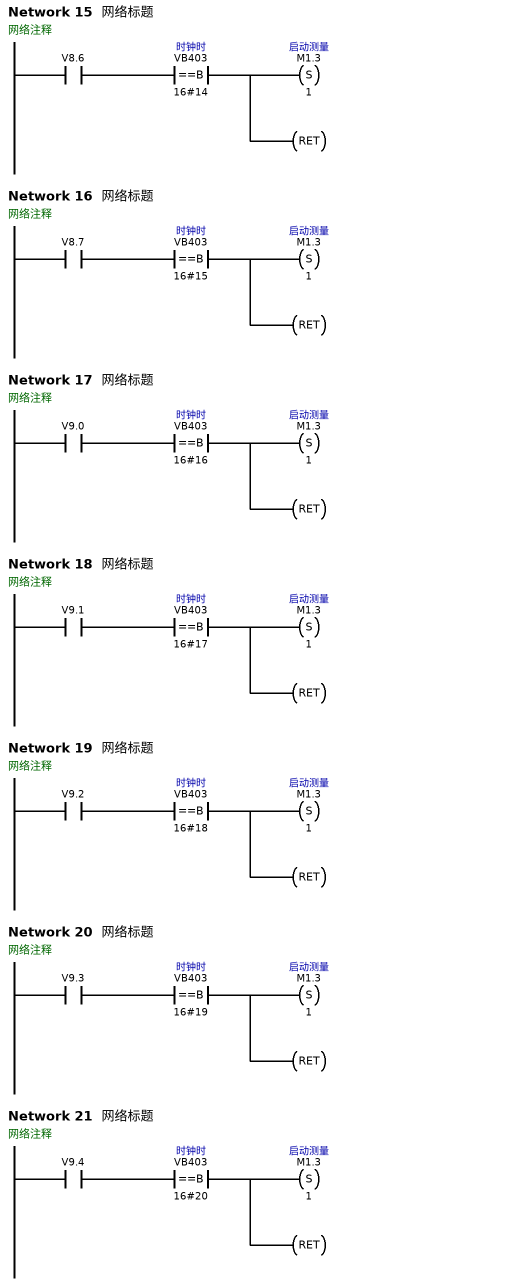
[picture p72: SBR13 networks 15-21]
Network 15 // 网络标题
// 网络注释
LD     V8.6
AB=    时钟时:VB403, 16#14
S      启动测量:M1.3, 1
CRET
Network 16 // 网络标题
// 网络注释
LD     V8.7
AB=    时钟时:VB403, 16#15
S      启动测量:M1.3, 1
CRET
Network 17 // 网络标题
// 网络注释
LD     V9.0
AB=    时钟时:VB403, 16#16
S      启动测量:M1.3, 1
CRET
Network 18 // 网络标题
// 网络注释
LD     V9.1
AB=    时钟时:VB403, 16#17
S      启动测量:M1.3, 1
CRET
Network 19 // 网络标题
// 网络注释
LD     V9.2
AB=    时钟时:VB403, 16#18
S      启动测量:M1.3, 1
CRET
Network 20 // 网络标题
// 网络注释
LD     V9.3
AB=    时钟时:VB403, 16#19
S      启动测量:M1.3, 1
CRET
Network 21 // 网络标题
// 网络注释
LD     V9.4
AB=    时钟时:VB403, 16#20
S      启动测量:M1.3, 1
CRET
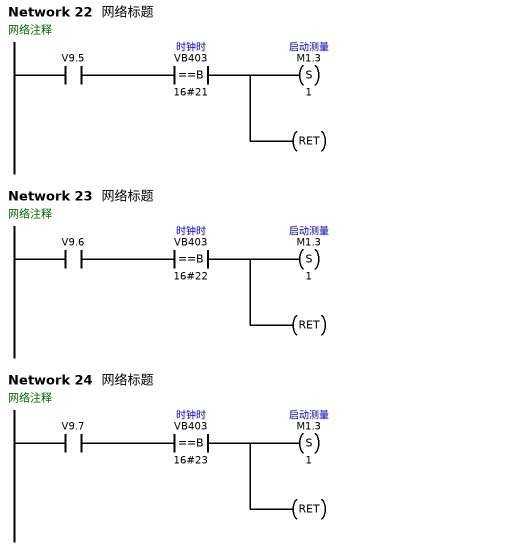
Network 22 // 网络标题
// 网络注释
LD     V9.5
AB=    时钟时:VB403, 16#21
S      启动测量:M1.3, 1
CRET
Network 23 // 网络标题
// 网络注释
LD     V9.6
AB=    时钟时:VB403, 16#22
S      启动测量:M1.3, 1
CRET
Network 24 // 网络标题
// 网络注释
LD     V9.7
AB=    时钟时:VB403, 16#23
S      启动测量:M1.3, 1
CRET
END_SUBROUTINE_BLOCK

SUBROUTINE_BLOCK Cal:SBR14
TITLE=子程序注释
VAR_INPUT
V:REAL;	// LD0 
Vo:REAL;	// LD4 
K:REAL;	// LD8 
b:REAL;	// LD12 
END_VAR
VAR_OUTPUT
吸光度:REAL;	// LD16 
值:REAL;	// LD20 
END_VAR
BEGIN
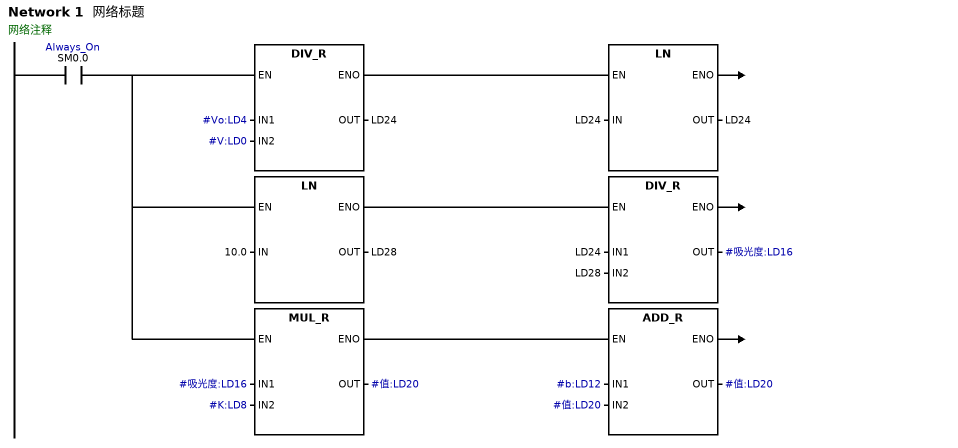
Network 1 // 网络标题
// 网络注释
LD     Always_On:SM0.0
LPS
MOVR   #Vo:LD4, LD24
AENO
/R     #V:LD0, LD24
AENO
LN     LD24, LD24
LRD
LN     10.0, LD28
AENO
MOVR   LD24, #吸光度:LD16
/R     LD28, #吸光度:LD16
LPP
MOVR   #吸光度:LD16, #值:LD20
AENO
*R     #K:LD8, #值:LD20
AENO
+R     #b:LD12, #值:LD20
END_SUBROUTINE_BLOCK

SUBROUTINE_BLOCK 偏离规则:SBR16
TITLE=子程序注释
VAR_INPUT
测量值:REAL;	// LD0 
标准值:REAL;	// LD4 
偏离比:REAL;	// LD8 0-100(10表示偏离百分之十以内视为通过)
END_VAR
VAR_OUTPUT
通过:BOOL;	// L12.0 
END_VAR
VAR
mid1:REAL;	// LD13 
mid2:REAL;	// LD17 
mid3:REAL;	// LD21 
上:REAL;	// LD25 
下:REAL;	// LD29 
END_VAR
BEGIN
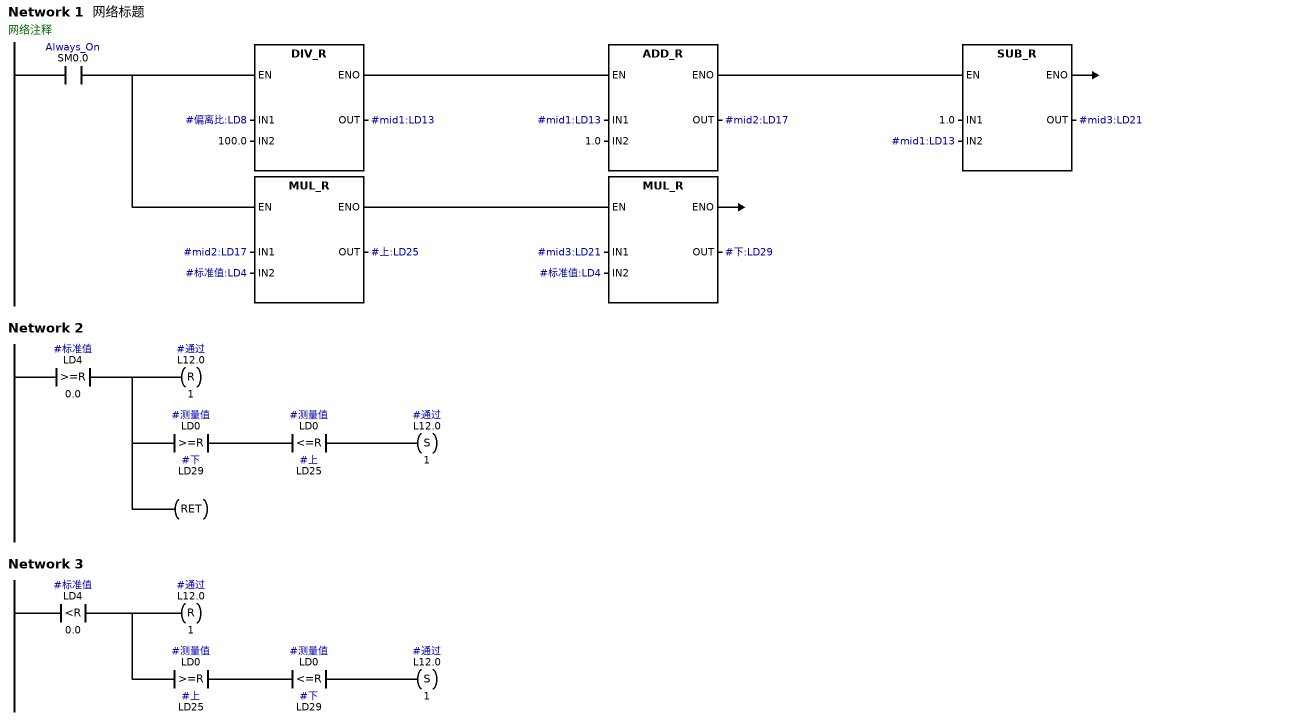
Network 1 // 网络标题
// 网络注释
LD     Always_On:SM0.0
LPS
MOVR   #偏离比:LD8, #mid1:LD13
AENO
/R     100.0, #mid1:LD13
AENO
MOVR   #mid1:LD13, #mid2:LD17
AENO
+R     1.0, #mid2:LD17
AENO
MOVR   1.0, #mid3:LD21
-R     #mid1:LD13, #mid3:LD21
LPP
MOVR   #mid2:LD17, #上:LD25
AENO
*R     #标准值:LD4, #上:LD25
AENO
MOVR   #mid3:LD21, #下:LD29
*R     #标准值:LD4, #下:LD29
Network 2
LDR>=  #标准值:LD4, 0.0
LPS
R      #通过:L12.0, 1
AR>=   #测量值:LD0, #下:LD29
AR<=   #测量值:LD0, #上:LD25
S      #通过:L12.0, 1
LPP
CRET
Network 3
LDR<   #标准值:LD4, 0.0
R      #通过:L12.0, 1
AR>=   #测量值:LD0, #上:LD25
AR<=   #测量值:LD0, #下:LD29
S      #通过:L12.0, 1
END_SUBROUTINE_BLOCK

SUBROUTINE_BLOCK 数据库:SBR17
TITLE=子程序注释
BEGIN
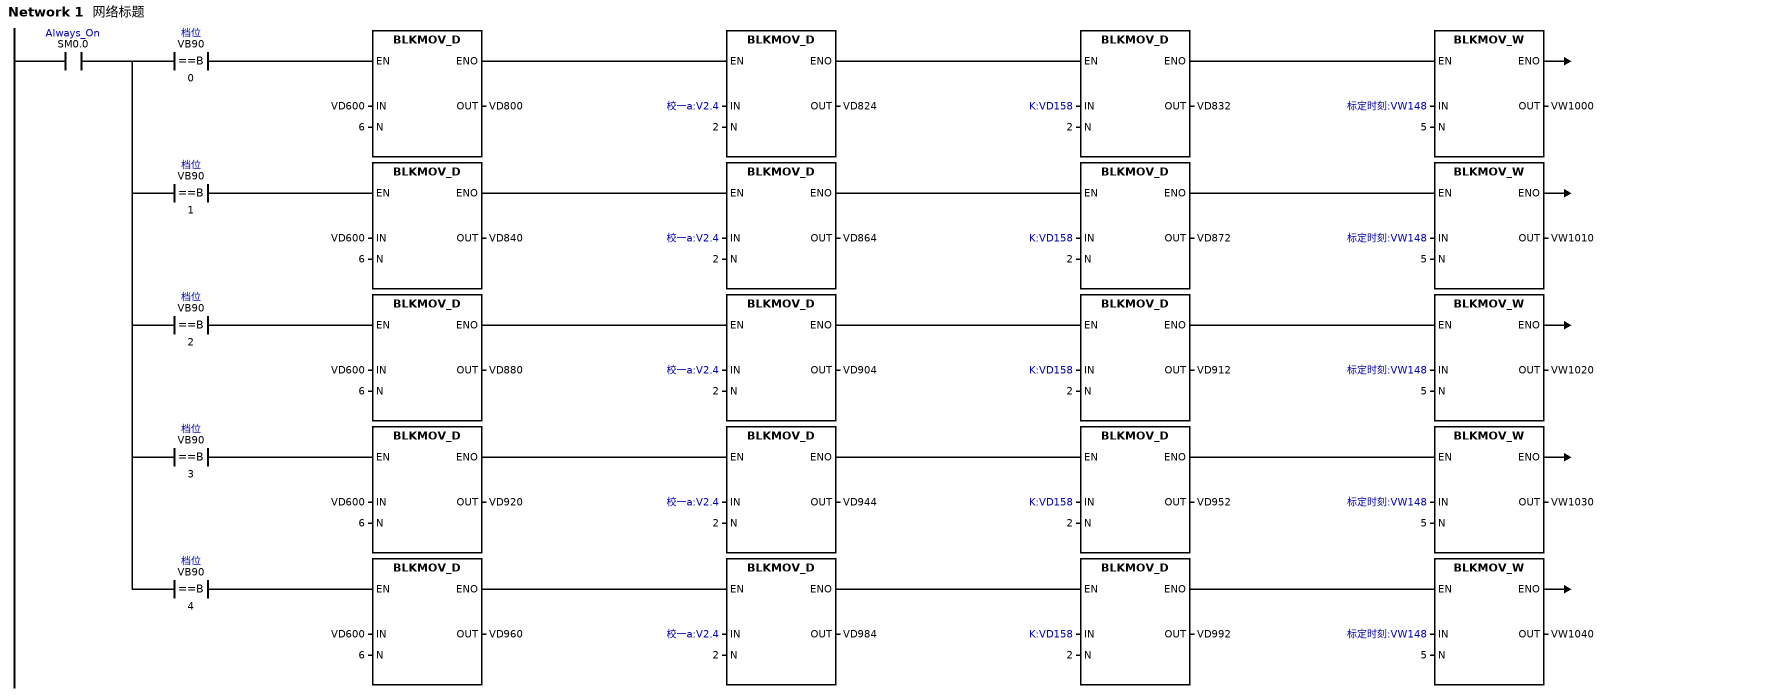
Network 1 // 网络标题
// (network saved uncompiled; LAD cells follow)
// row 0: c0 -| |- Always_On:SM0.0 v  c1 -|==B|- 档位:VB90, 0  c2 --  c3 [BLKMOV_D EN:=power@row0, IN:=VD600, N:=6, ENO=>power, OUT=>VD800]  c4 --  c5 --  c6 [BLKMOV_D EN:=power@row0, IN:=校一a:V2.4, N:=2, ENO=>power, OUT=>VD824]  c7 --  c8 --  c9 [BLKMOV_D EN:=power@row0, IN:=K:VD158, N:=2, ENO=>power, OUT=>VD832]  c10 --  c11 --  c12 [BLKMOV_W EN:=power@row0, IN:=标定时刻:VW148, N:=5, ENO=>power, OUT=>VW1000]  c13 ->
// row 1: c0 ^v  c3 [box]  c6 [box]  c9 [box]  c12 [box]
// row 2: c0 ^v  c1 -|==B|- 档位:VB90, 1  c2 --  c3 [BLKMOV_D EN:=power@row2, IN:=VD600, N:=6, ENO=>power, OUT=>VD840]  c4 --  c5 --  c6 [BLKMOV_D EN:=power@row2, IN:=校一a:V2.4, N:=2, ENO=>power, OUT=>VD864]  c7 --  c8 --  c9 [BLKMOV_D EN:=power@row2, IN:=K:VD158, N:=2, ENO=>power, OUT=>VD872]  c10 --  c11 --  c12 [BLKMOV_W EN:=power@row2, IN:=标定时刻:VW148, N:=5, ENO=>power, OUT=>VW1010]  c13 ->
// row 3: c0 ^v  c3 [box]  c6 [box]  c9 [box]  c12 [box]
// row 4: c0 ^v  c1 -|==B|- 档位:VB90, 2  c2 --  c3 [BLKMOV_D EN:=power@row4, IN:=VD600, N:=6, ENO=>power, OUT=>VD880]  c4 --  c5 --  c6 [BLKMOV_D EN:=power@row4, IN:=校一a:V2.4, N:=2, ENO=>power, OUT=>VD904]  c7 --  c8 --  c9 [BLKMOV_D EN:=power@row4, IN:=K:VD158, N:=2, ENO=>power, OUT=>VD912]  c10 --  c11 --  c12 [BLKMOV_W EN:=power@row4, IN:=标定时刻:VW148, N:=5, ENO=>power, OUT=>VW1020]  c13 ->
// row 5: c0 ^v  c3 [box]  c6 [box]  c9 [box]  c12 [box]
// row 6: c0 ^v  c1 -|==B|- 档位:VB90, 3  c2 --  c3 [BLKMOV_D EN:=power@row6, IN:=VD600, N:=6, ENO=>power, OUT=>VD920]  c4 --  c5 --  c6 [BLKMOV_D EN:=power@row6, IN:=校一a:V2.4, N:=2, ENO=>power, OUT=>VD944]  c7 --  c8 --  c9 [BLKMOV_D EN:=power@row6, IN:=K:VD158, N:=2, ENO=>power, OUT=>VD952]  c10 --  c11 --  c12 [BLKMOV_W EN:=power@row6, IN:=标定时刻:VW148, N:=5, ENO=>power, OUT=>VW1030]  c13 ->
// row 7: c0 ^v  c3 [box]  c6 [box]  c9 [box]  c12 [box]
// row 8: c0 ^  c1 -|==B|- 档位:VB90, 4  c2 --  c3 [BLKMOV_D EN:=power@row8, IN:=VD600, N:=6, ENO=>power, OUT=>VD960]  c4 --  c5 --  c6 [BLKMOV_D EN:=power@row8, IN:=校一a:V2.4, N:=2, ENO=>power, OUT=>VD984]  c7 --  c8 --  c9 [BLKMOV_D EN:=power@row8, IN:=K:VD158, N:=2, ENO=>power, OUT=>VD992]  c10 --  c11 --  c12 [BLKMOV_W EN:=power@row8, IN:=标定时刻:VW148, N:=5, ENO=>power, OUT=>VW1040]  c13 ->
// row 9: c3 [box]  c6 [box]  c9 [box]  c12 [box]
END_SUBROUTINE_BLOCK

SUBROUTINE_BLOCK 换挡:SBR19
TITLE=每个切换范围包含高低两个档位，当前处于低档则切换到高档，反之亦然
BEGIN
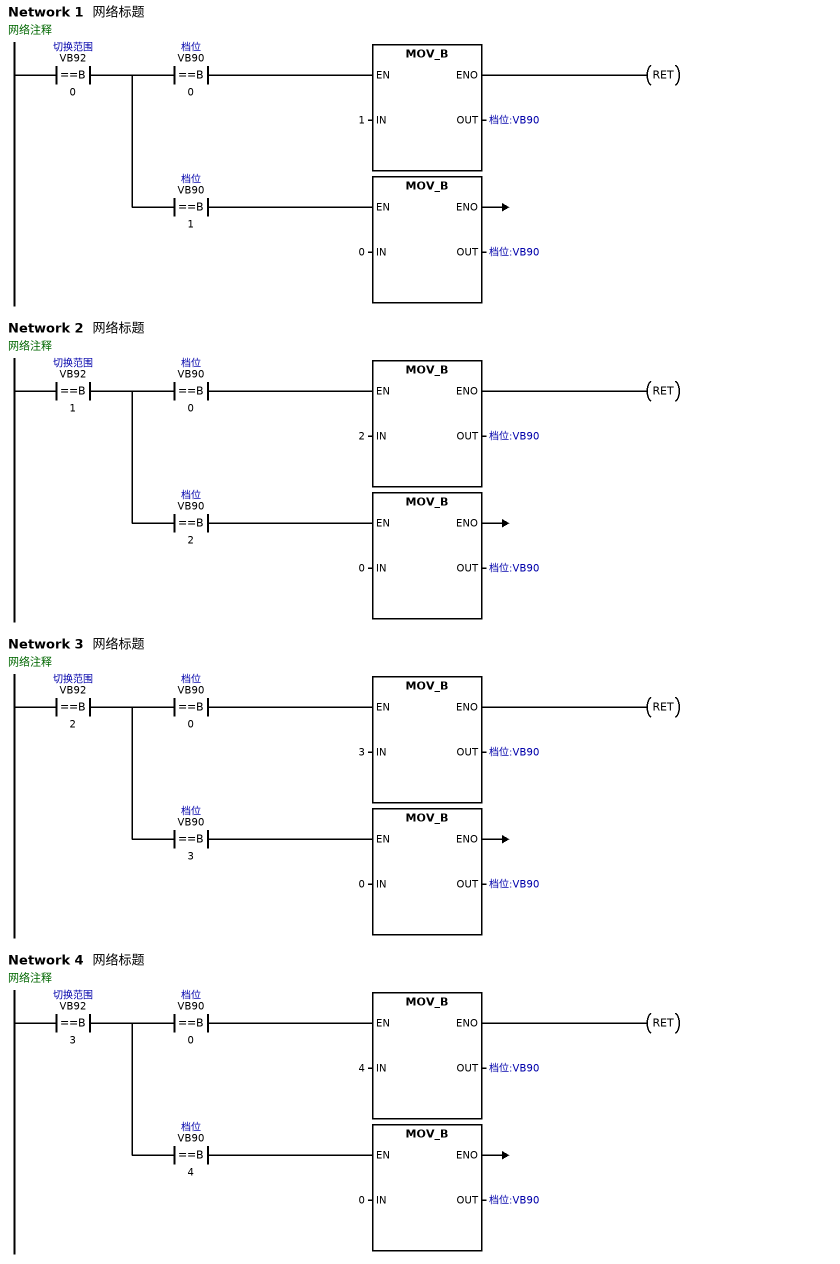
Network 1 // 网络标题
// 网络注释
LDB=   切换范围:VB92, 0
LPS
AB=    档位:VB90, 0
MOVB   1, 档位:VB90
AENO
CRET
LPP
AB=    档位:VB90, 1
MOVB   0, 档位:VB90
Network 2 // 网络标题
// 网络注释
LDB=   切换范围:VB92, 1
LPS
AB=    档位:VB90, 0
MOVB   2, 档位:VB90
AENO
CRET
LPP
AB=    档位:VB90, 2
MOVB   0, 档位:VB90
Network 3 // 网络标题
// 网络注释
LDB=   切换范围:VB92, 2
LPS
AB=    档位:VB90, 0
MOVB   3, 档位:VB90
AENO
CRET
LPP
AB=    档位:VB90, 3
MOVB   0, 档位:VB90
Network 4 // 网络标题
// 网络注释
LDB=   切换范围:VB92, 3
LPS
AB=    档位:VB90, 0
MOVB   4, 档位:VB90
AENO
CRET
LPP
AB=    档位:VB90, 4
MOVB   0, 档位:VB90
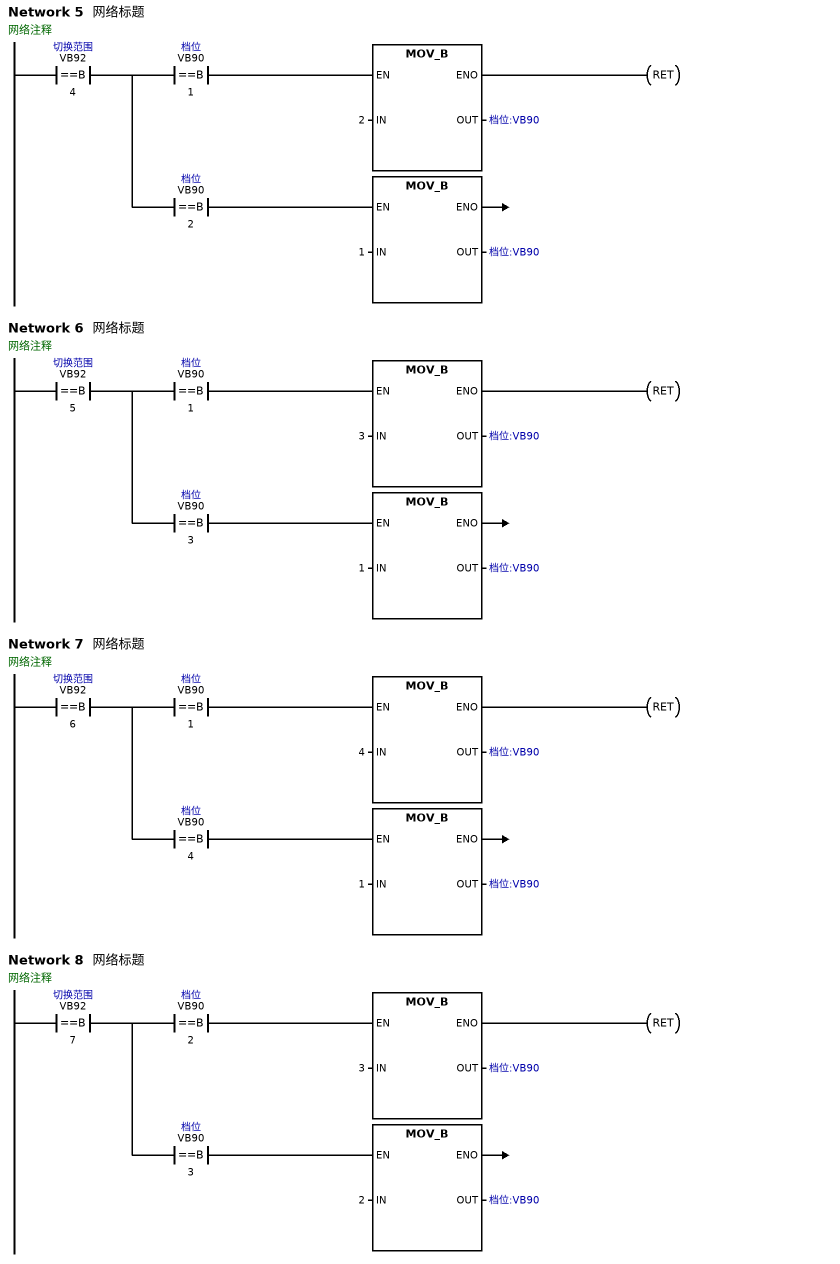
Network 5 // 网络标题
// 网络注释
LDB=   切换范围:VB92, 4
LPS
AB=    档位:VB90, 1
MOVB   2, 档位:VB90
AENO
CRET
LPP
AB=    档位:VB90, 2
MOVB   1, 档位:VB90
Network 6 // 网络标题
// 网络注释
LDB=   切换范围:VB92, 5
LPS
AB=    档位:VB90, 1
MOVB   3, 档位:VB90
AENO
CRET
LPP
AB=    档位:VB90, 3
MOVB   1, 档位:VB90
Network 7 // 网络标题
// 网络注释
LDB=   切换范围:VB92, 6
LPS
AB=    档位:VB90, 1
MOVB   4, 档位:VB90
AENO
CRET
LPP
AB=    档位:VB90, 4
MOVB   1, 档位:VB90
Network 8 // 网络标题
// 网络注释
LDB=   切换范围:VB92, 7
LPS
AB=    档位:VB90, 2
MOVB   3, 档位:VB90
AENO
CRET
LPP
AB=    档位:VB90, 3
MOVB   2, 档位:VB90
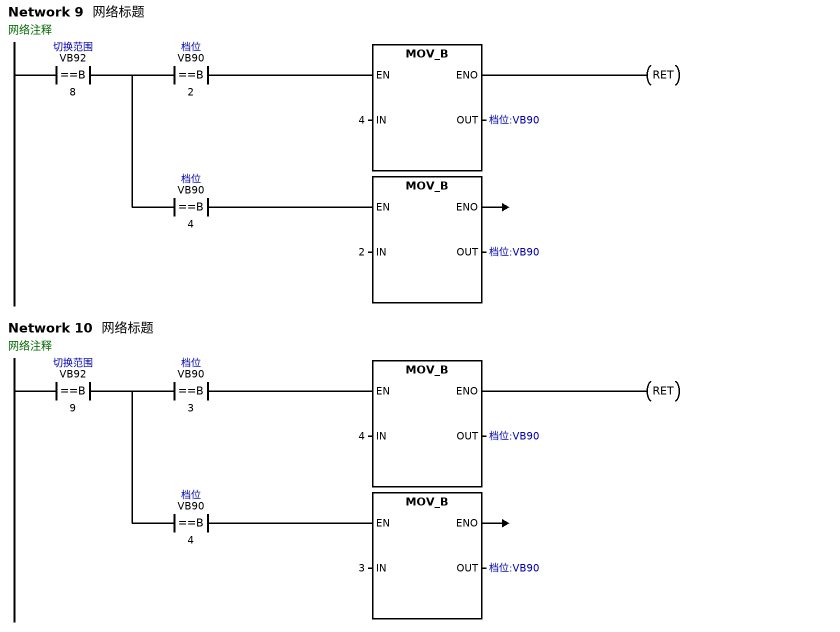
Network 9 // 网络标题
// 网络注释
LDB=   切换范围:VB92, 8
LPS
AB=    档位:VB90, 2
MOVB   4, 档位:VB90
AENO
CRET
LPP
AB=    档位:VB90, 4
MOVB   2, 档位:VB90
Network 10 // 网络标题
// 网络注释
LDB=   切换范围:VB92, 9
LPS
AB=    档位:VB90, 3
MOVB   4, 档位:VB90
AENO
CRET
LPP
AB=    档位:VB90, 4
MOVB   3, 档位:VB90
END_SUBROUTINE_BLOCK

// SBR21: protected block, not included

SUBROUTINE_BLOCK ReCal:SBR22
TITLE=子程序注释
VAR_INPUT
Uo:REAL;	// LD0 
C‘:REAL;	// LD4 
K:REAL;	// LD8 
b:REAL;	// LD12 
END_VAR
VAR_OUTPUT
U‘:REAL;	// LD16 
A’:REAL;	// LD20 
END_VAR
VAR
mid:REAL;	// LD24 
END_VAR
BEGIN
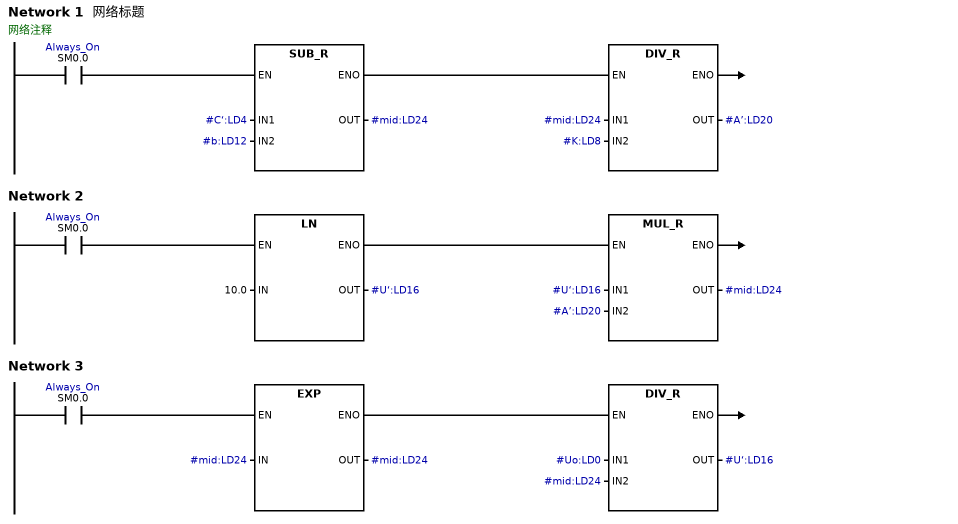
Network 1 // 网络标题
// 网络注释
LD     Always_On:SM0.0
MOVR   #C‘:LD4, #mid:LD24
AENO
-R     #b:LD12, #mid:LD24
AENO
MOVR   #mid:LD24, #A’:LD20
/R     #K:LD8, #A’:LD20
Network 2
LD     Always_On:SM0.0
LN     10.0, #U‘:LD16
AENO
MOVR   #U‘:LD16, #mid:LD24
*R     #A’:LD20, #mid:LD24
Network 3
LD     Always_On:SM0.0
EXP    #mid:LD24, #mid:LD24
AENO
MOVR   #Uo:LD0, #U‘:LD16
/R     #mid:LD24, #U‘:LD16
Network 4 // 网络标题
// 网络注释
END_SUBROUTINE_BLOCK

SUBROUTINE_BLOCK 标准R_I:SBR23
TITLE=子程序注释
VAR_INPUT
R_H:REAL;	// LD0 
R_L:REAL;	// LD4 
I_H:WORD;	// LW8 
I_L:WORD;	// LW10 
Input:REAL;	// LD12 
END_VAR
VAR_OUTPUT
output:WORD;	// LW16 
END_VAR
BEGIN
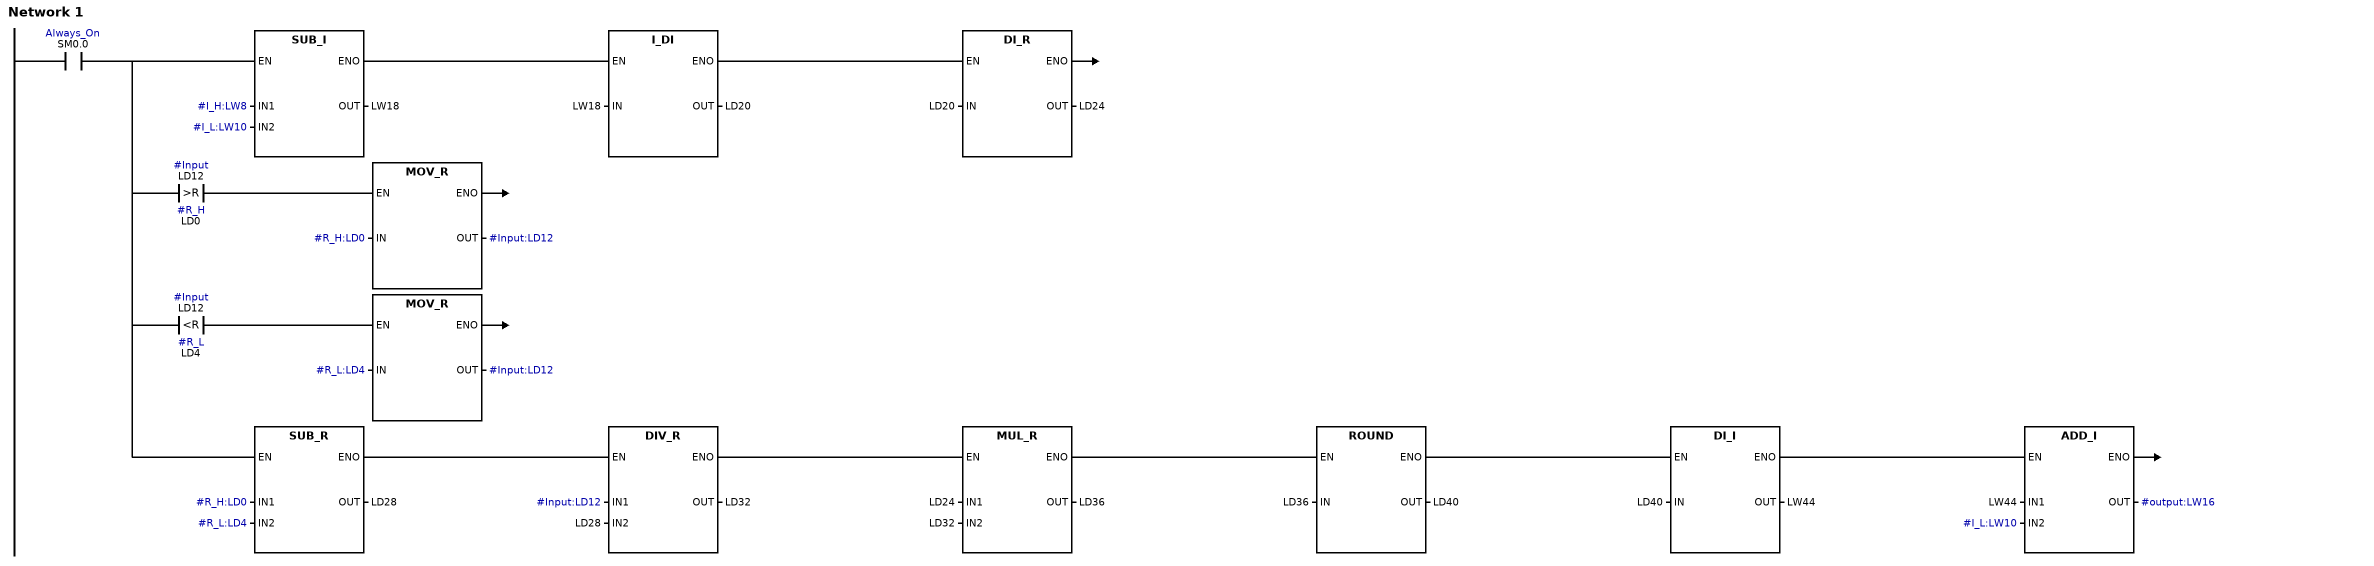
Network 1
LD     Always_On:SM0.0
LPS
MOVW   #I_H:LW8, LW18
AENO
-I     #I_L:LW10, LW18
AENO
ITD    LW18, LD20
AENO
DTR    LD20, LD24
LRD
AR>    #Input:LD12, #R_H:LD0
MOVR   #R_H:LD0, #Input:LD12
LRD
AR<    #Input:LD12, #R_L:LD4
MOVR   #R_L:LD4, #Input:LD12
LPP
MOVR   #R_H:LD0, LD28
AENO
-R     #R_L:LD4, LD28
AENO
MOVR   #Input:LD12, LD32
AENO
/R     LD28, LD32
AENO
MOVR   LD24, LD36
AENO
*R     LD32, LD36
AENO
ROUND  LD36, LD40
AENO
DTI    LD40, LW44
AENO
MOVW   LW44, #output:LW16
+I     #I_L:LW10, #output:LW16
END_SUBROUTINE_BLOCK

SUBROUTINE_BLOCK 动态管控参数:SBR24
TITLE=子程序注释
BEGIN
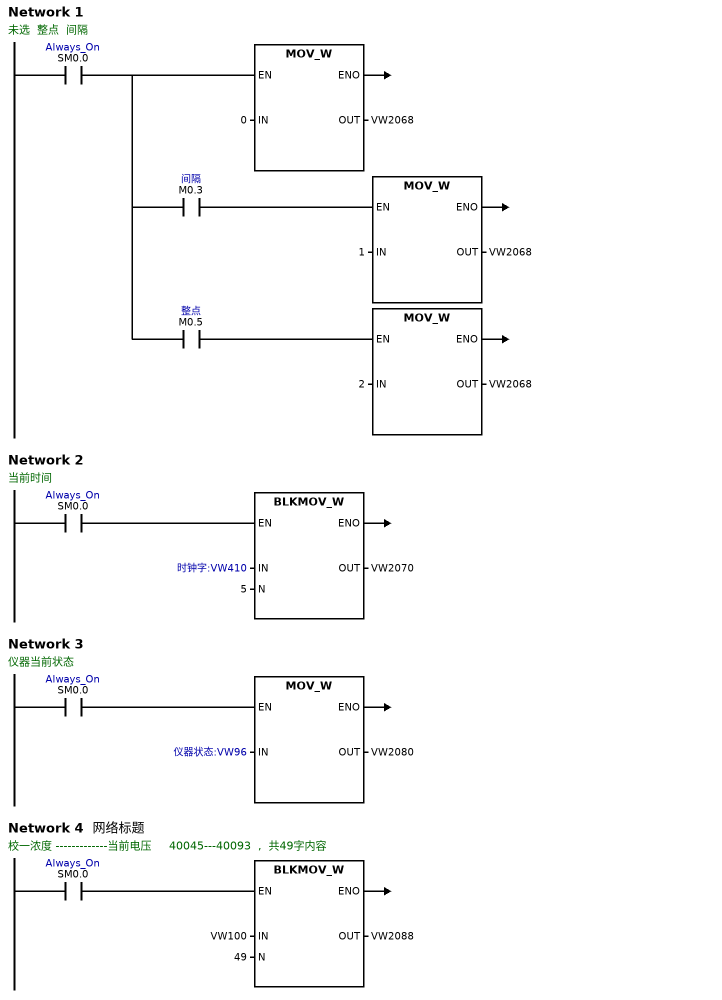
Network 1
//  未选  整点  间隔
LD     Always_On:SM0.0
LPS
MOVW   0, VW2068
A      间隔:M0.3
MOVW   1, VW2068
LPP
A      整点:M0.5
MOVW   2, VW2068
Network 2
// 当前时间
LD     Always_On:SM0.0
BMW    时钟字:VW410, VW2070, 5
Network 3
// 仪器当前状态
LD     Always_On:SM0.0
MOVW   仪器状态:VW96, VW2080
Network 4 // 网络标题
// 校一浓度 -------------当前电压     40045---40093  ,  共49字内容
LD     Always_On:SM0.0
BMW    VW100, VW2088, 49
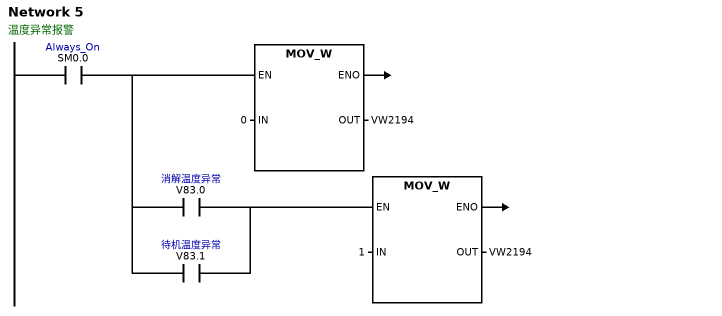
Network 5
// 温度异常报警
LD     Always_On:SM0.0
MOVW   0, VW2194
LD     消解温度异常:V83.0
O      待机温度异常:V83.1
ALD
MOVW   1, VW2194
Network 6
// 电极电压异常报警
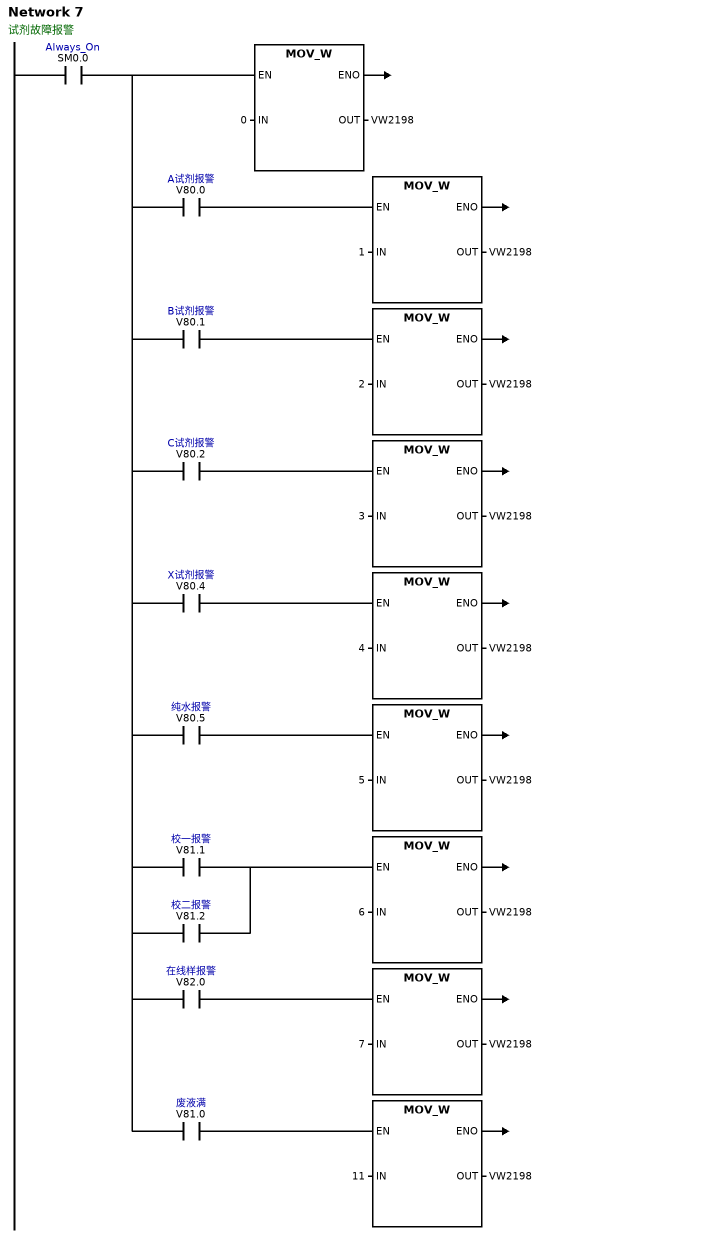
Network 7
// 试剂故障报警
LD     Always_On:SM0.0
LPS
MOVW   0, VW2198
A      A试剂报警:V80.0
MOVW   1, VW2198
LRD
A      B试剂报警:V80.1
MOVW   2, VW2198
LRD
A      C试剂报警:V80.2
MOVW   3, VW2198
LRD
A      X试剂报警:V80.4
MOVW   4, VW2198
LRD
A      纯水报警:V80.5
MOVW   5, VW2198
LRD
LD     校一报警:V81.1
O      校二报警:V81.2
ALD
MOVW   6, VW2198
LPP
LPS
A      在线样报警:V82.0
MOVW   7, VW2198
LPP
A      废液满:V81.0
MOVW   11, VW2198
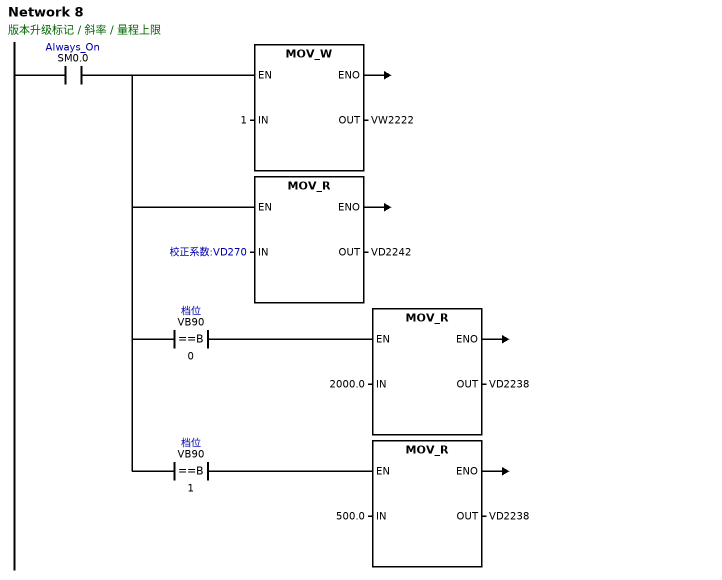
Network 8
// 版本升级标记
// 斜率
// 量程上限
LD     Always_On:SM0.0
LPS
MOVW   1, VW2222
MOVR   校正系数:VD270, VD2242
AB=    档位:VB90, 0
MOVR   2000.0, VD2238
LPP
AB=    档位:VB90, 1
MOVR   500.0, VD2238
END_SUBROUTINE_BLOCK

SUBROUTINE_BLOCK 设备状态:SBR25
TITLE=子程序注释
BEGIN
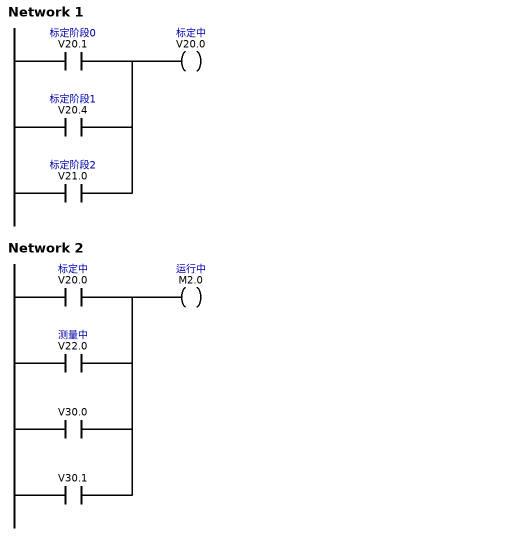
Network 1
LD     标定阶段0:V20.1
O      标定阶段1:V20.4
O      标定阶段2:V21.0
=      标定中:V20.0
Network 2
LD     标定中:V20.0
O      测量中:V22.0
O      V30.0
O      V30.1
=      运行中:M2.0
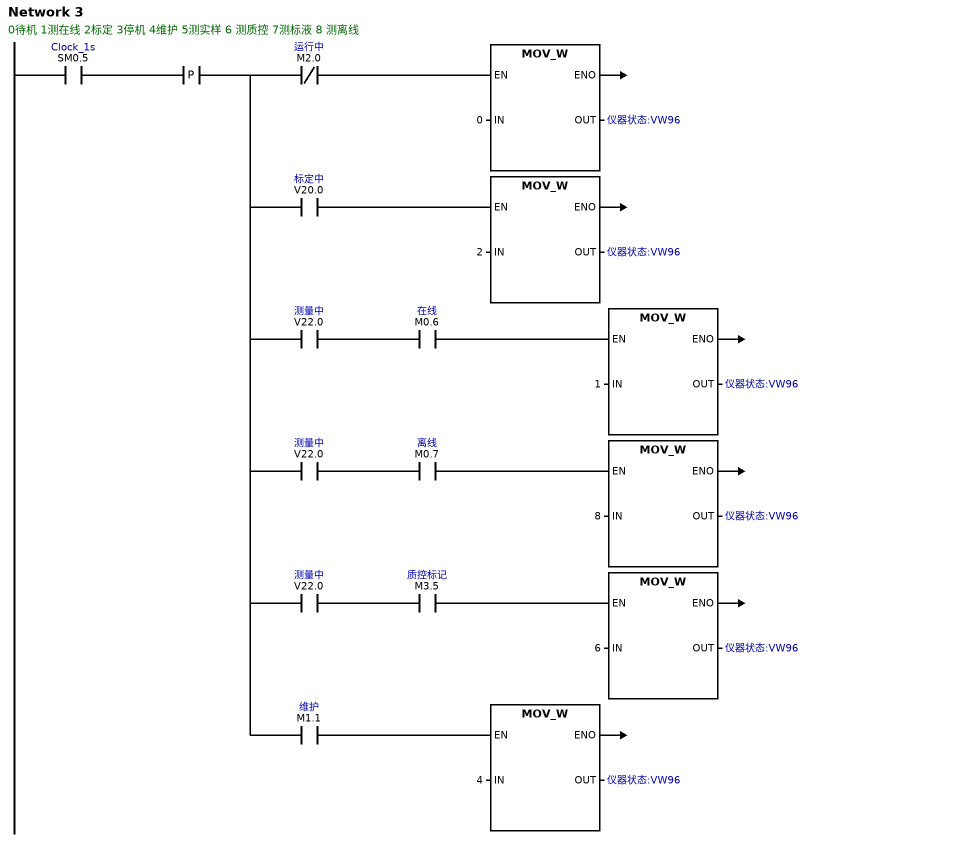
Network 3
// 0待机 1测在线 2标定 3停机 4维护 5测实样 6 测质控 7测标液 8 测离线
LD     Clock_1s:SM0.5
EU
LPS
AN     运行中:M2.0
MOVW   0, 仪器状态:VW96
LRD
A      标定中:V20.0
MOVW   2, 仪器状态:VW96
LRD
A      测量中:V22.0
A      在线:M0.6
MOVW   1, 仪器状态:VW96
LRD
A      测量中:V22.0
A      离线:M0.7
MOVW   8, 仪器状态:VW96
LRD
A      测量中:V22.0
A      质控标记:M3.5
MOVW   6, 仪器状态:VW96
LPP
A      维护:M1.1
MOVW   4, 仪器状态:VW96
END_SUBROUTINE_BLOCK

SUBROUTINE_BLOCK 密码:SBR26
TITLE=子程序注释
BEGIN
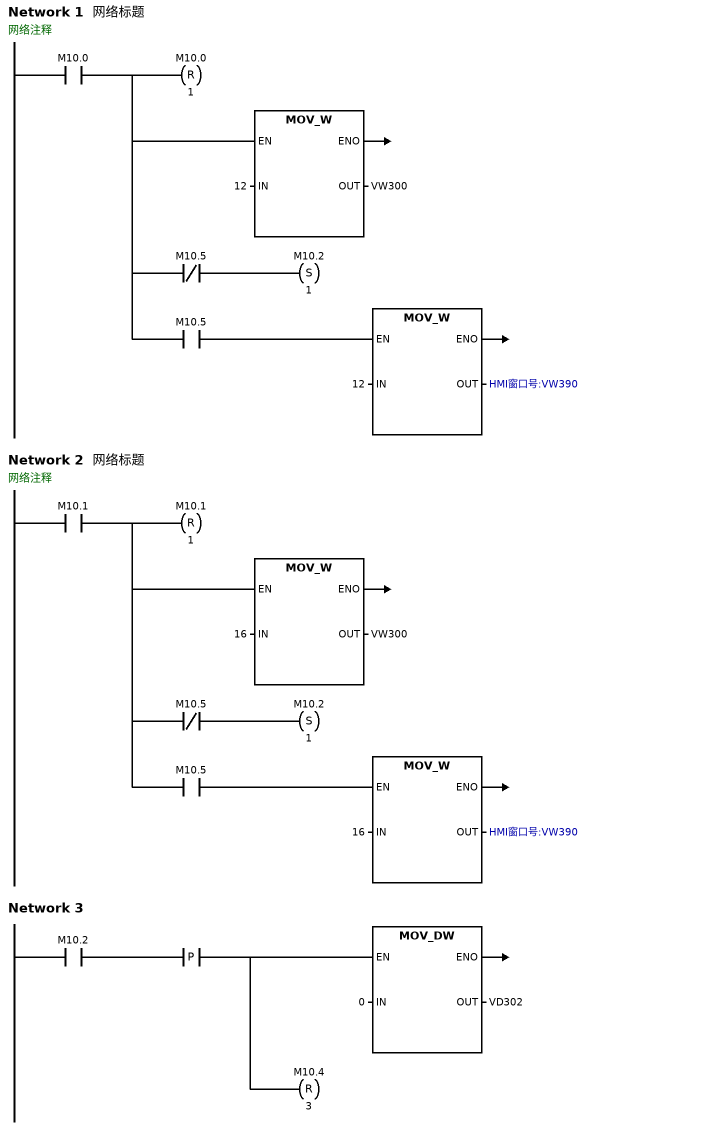
Network 1 // 网络标题
// 网络注释
LD     M10.0
LPS
R      M10.0, 1
MOVW   12, VW300
AN     M10.5
S      M10.2, 1
LPP
A      M10.5
MOVW   12, HMI窗口号:VW390
Network 2 // 网络标题
// 网络注释
LD     M10.1
LPS
R      M10.1, 1
MOVW   16, VW300
AN     M10.5
S      M10.2, 1
LPP
A      M10.5
MOVW   16, HMI窗口号:VW390
Network 3
LD     M10.2
EU
MOVD   0, VD302
R      M10.4, 3
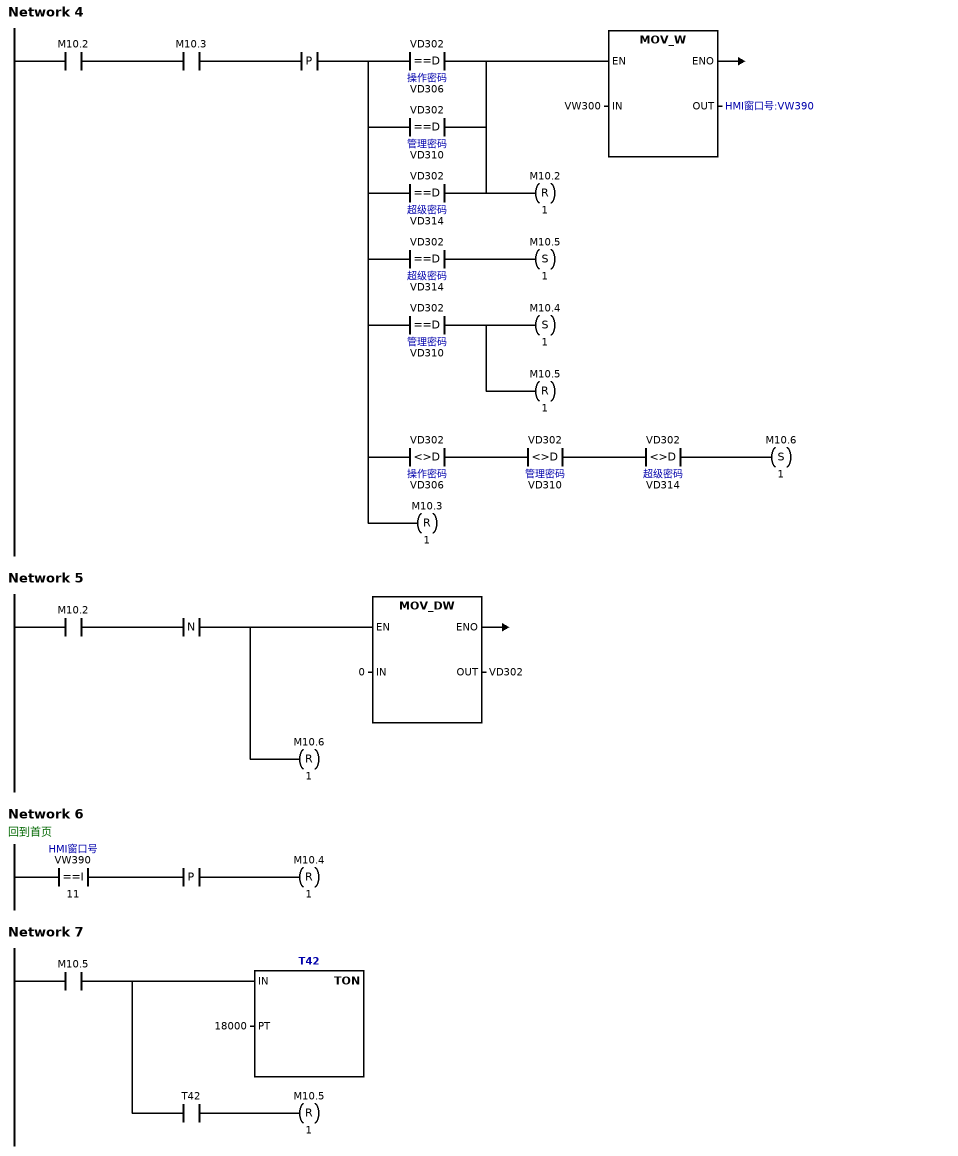
Network 4
LD     M10.2
A      M10.3
EU
LPS
LDD=   VD302, 操作密码:VD306
OD=    VD302, 管理密码:VD310
OD=    VD302, 超级密码:VD314
ALD
MOVW   VW300, HMI窗口号:VW390
R      M10.2, 1
LRD
AD=    VD302, 超级密码:VD314
S      M10.5, 1
LRD
AD=    VD302, 管理密码:VD310
S      M10.4, 1
R      M10.5, 1
LPP
LPS
AD<>   VD302, 操作密码:VD306
AD<>   VD302, 管理密码:VD310
AD<>   VD302, 超级密码:VD314
S      M10.6, 1
LPP
R      M10.3, 1
Network 5
LD     M10.2
ED
MOVD   0, VD302
R      M10.6, 1
Network 6
// 回到首页
LDW=   HMI窗口号:VW390, 11
EU
R      M10.4, 1
Network 7
LD     M10.5
TON    T42, 18000
A      T42
R      M10.5, 1
END_SUBROUTINE_BLOCK

SUBROUTINE_BLOCK 单位转换:SBR27
TITLE=子程序注释
BEGIN
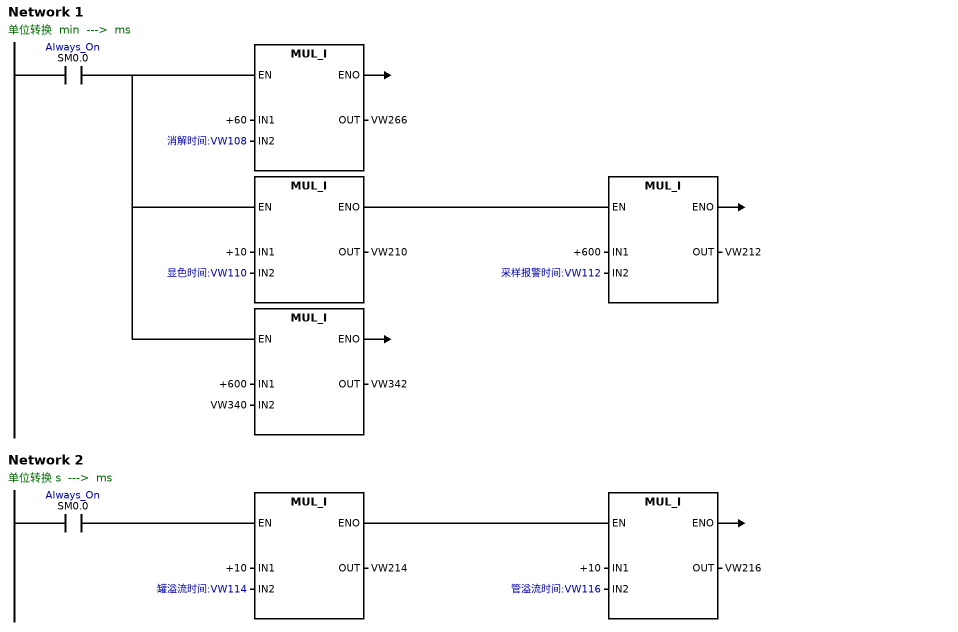
Network 1
// 单位转换  min  --->  ms
LD     Always_On:SM0.0
LPS
MOVW   +60, VW266
*I     消解时间:VW108, VW266
MOVW   +10, VW210
AENO
*I     显色时间:VW110, VW210
AENO
MOVW   +600, VW212
*I     采样报警时间:VW112, VW212
LPP
MOVW   +600, VW342
*I     VW340, VW342
Network 2
// 单位转换 s  --->  ms
LD     Always_On:SM0.0
MOVW   +10, VW214
AENO
*I     罐溢流时间:VW114, VW214
AENO
MOVW   +10, VW216
*I     管溢流时间:VW116, VW216
Network 3 // 网络标题
// 网络注释
END_SUBROUTINE_BLOCK

SUBROUTINE_BLOCK 读时钟:SBR28
TITLE=
BEGIN
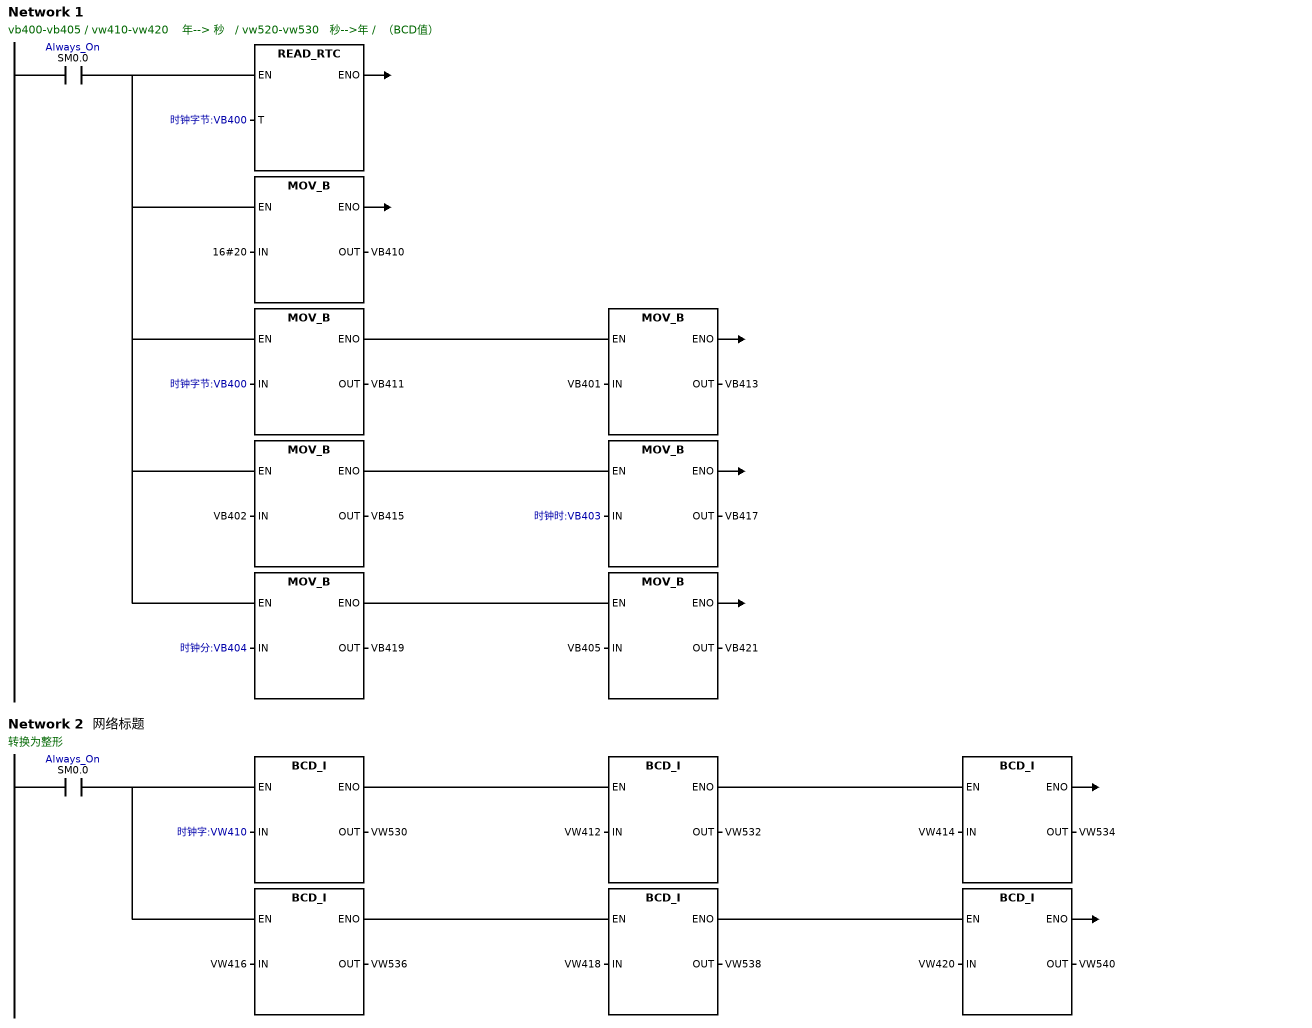
Network 1
// vb400-vb405
// vw410-vw420    年--> 秒  
// vw520-vw530   秒-->年
//  （BCD值）
LD     Always_On:SM0.0
LPS
TODR   时钟字节:VB400
MOVB   16#20, VB410
MOVB   时钟字节:VB400, VB411
AENO
MOVB   VB401, VB413
LRD
MOVB   VB402, VB415
AENO
MOVB   时钟时:VB403, VB417
LPP
MOVB   时钟分:VB404, VB419
AENO
MOVB   VB405, VB421
Network 2 // 网络标题
// 转换为整形
LD     Always_On:SM0.0
LPS
MOVW   时钟字:VW410, VW530
AENO
BCDI   VW530
AENO
MOVW   VW412, VW532
AENO
BCDI   VW532
AENO
MOVW   VW414, VW534
BCDI   VW534
LPP
MOVW   VW416, VW536
AENO
BCDI   VW536
AENO
MOVW   VW418, VW538
AENO
BCDI   VW538
AENO
MOVW   VW420, VW540
BCDI   VW540
END_SUBROUTINE_BLOCK

SUBROUTINE_BLOCK M7抽推比色皿:SBR29
TITLE=
VAR_INPUT
抽:BOOL;	// L0.0 
时间:WORD;	// LW1 
END_VAR
VAR_IN_OUT
启动位:BOOL;	// L3.0 
END_VAR
VAR_OUTPUT
结束位:BOOL;	// L3.1 
END_VAR
BEGIN
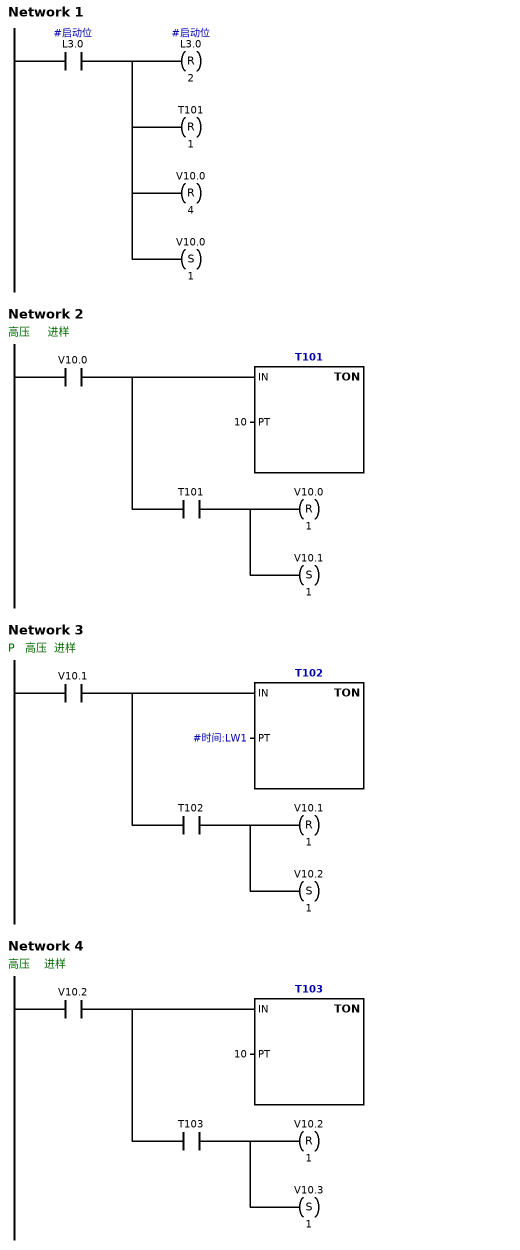
Network 1
LD     #启动位:L3.0
R      #启动位:L3.0, 2
R      T101, 1
R      V10.0, 4
S      V10.0, 1
Network 2
// 高压     进样
LD     V10.0
TON    T101, 10
A      T101
R      V10.0, 1
S      V10.1, 1
Network 3
// P   高压  进样
LD     V10.1
TON    T102, #时间:LW1
A      T102
R      V10.1, 1
S      V10.2, 1
Network 4
// 高压    进样
LD     V10.2
TON    T103, 10
A      T103
R      V10.2, 1
S      V10.3, 1
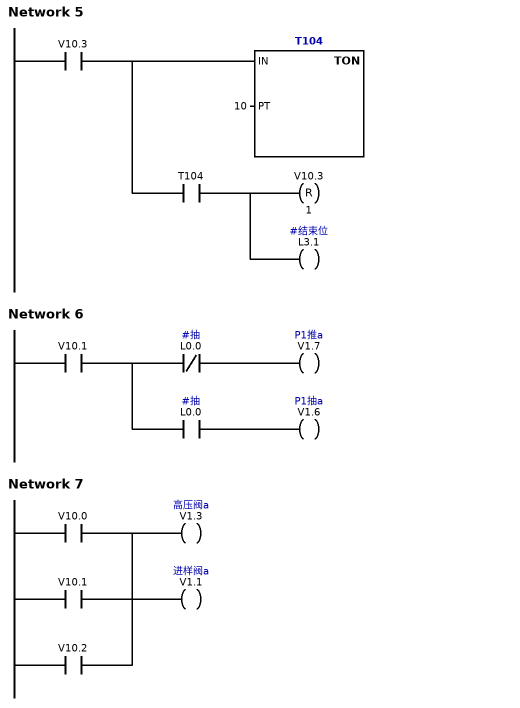
Network 5
LD     V10.3
TON    T104, 10
A      T104
R      V10.3, 1
=      #结束位:L3.1
Network 6
LD     V10.1
LPS
AN     #抽:L0.0
=      P1推a:V1.7
LPP
A      #抽:L0.0
=      P1抽a:V1.6
Network 7
LD     V10.0
O      V10.1
O      V10.2
=      高压阀a:V1.3
=      进样阀a:V1.1
Network 8 // 网络标题
// 网络注释
END_SUBROUTINE_BLOCK

// SBR30: protected block, not included

// SBR31: protected block, not included

// SBR32: protected block, not included

SUBROUTINE_BLOCK M8抽推多联体:SBR33
TITLE=
VAR_INPUT
抽:BOOL;	// L0.0 
时间:WORD;	// LW1 
END_VAR
VAR_IN_OUT
启动位:BOOL;	// L3.0 
END_VAR
VAR_OUTPUT
结束位:BOOL;	// L3.1 
阀:BOOL;	// L3.2 
END_VAR
BEGIN
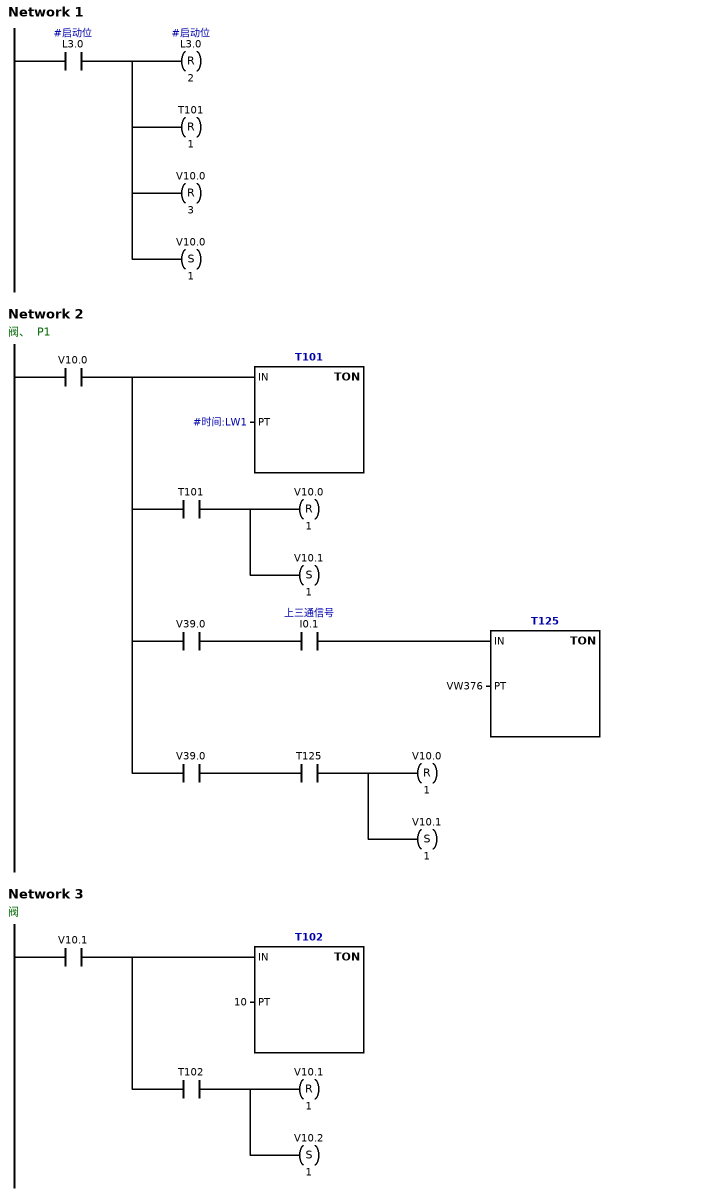
Network 1
LD     #启动位:L3.0
R      #启动位:L3.0, 2
R      T101, 1
R      V10.0, 3
S      V10.0, 1
Network 2
// 阀、  P1
LD     V10.0
LPS
TON    T101, #时间:LW1
A      T101
R      V10.0, 1
S      V10.1, 1
LRD
A      V39.0
A      上三通信号:I0.1
TON    T125, VW376
LPP
A      V39.0
A      T125
R      V10.0, 1
S      V10.1, 1
Network 3
// 阀
LD     V10.1
TON    T102, 10
A      T102
R      V10.1, 1
S      V10.2, 1
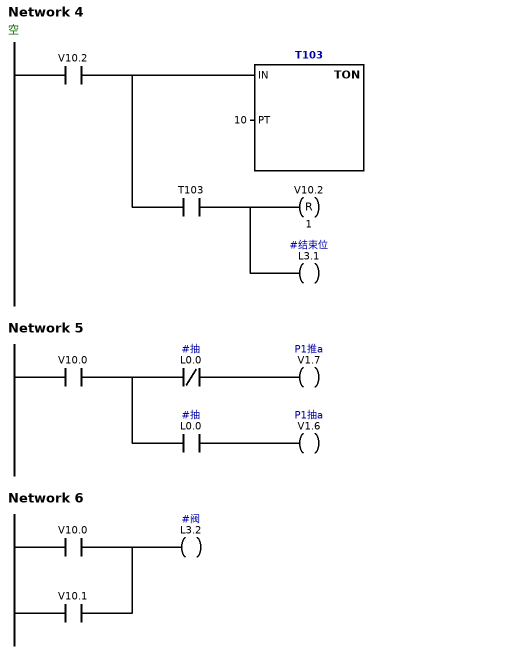
Network 4
// 空
LD     V10.2
TON    T103, 10
A      T103
R      V10.2, 1
=      #结束位:L3.1
Network 5
LD     V10.0
LPS
AN     #抽:L0.0
=      P1推a:V1.7
LPP
A      #抽:L0.0
=      P1抽a:V1.6
Network 6
LD     V10.0
O      V10.1
=      #阀:L3.2
Network 7 // 网络标题
// 网络注释
END_SUBROUTINE_BLOCK

SUBROUTINE_BLOCK 复位:SBR34
TITLE=级别越高复位内容越多
VAR_INPUT
level:BYTE;	// LB0 
END_VAR
BEGIN
